// TIA Portal project "S7-1500 ile GELİŞMİŞ Tavuk Çiftliği" (V18)

(* hardware
DEVICE "S7-1500/ET200MP station_1"  S7-1500 station
   slot 0: "Rail_0"  Rack  6ES7 590-1***0-0AA0
   slot 1: "PLC_1"  CPU 1512C-1 PN  6ES7 512-1CK01-0AB0  V2.8
      slot 3: "CPU display_1"  6ES7591-1AA00-0AA0
      slot 32768: "PROFINET interface_1"  X1
         slot 32769: "Port_1"  X1 P1
         slot 32770: "Port_2"  X1 P2
      slot 34817: "Virtual CP interface port_1"  Virtual CP interface port  Virtual CP interface port
DEVICE "HMI_1"  KTP700 Basic PN
   slot 0: "HMI_1"  KTP700 Basic PN  6AV2 123-2GB03-0AX0  14.0.1.0
   slot 1: "HMI_RT_1"  KTP700 Basic PN  6AV2 123-2GB03-0AX0  14.0.1.0
   slot 5: "HMI_1.IE_CP_1"  PROFINET Interface  14.0.1.0
      slot 1: "PROFINET Interface_1"  PROFINET Interface
         slot 1: "Port_1"  Port
*)

// ===== PLC "PLC_1"  CPU 1512C-1 PN =====

VAR_GLOBAL   // PLC tag table "Default tag table"
   "Analog Giriş" AT %IW126 : Word;
   "Kış" AT %I0.1 : Bool;
   "Yaz" AT %I0.2 : Bool;
   "Reset" AT %I0.0 : Bool;
   "Isıtıcı" AT %Q0.1 : Bool;
   "Soğutucu" AT %Q0.2 : Bool;
   "Tag_1" AT %Q0.0 : Bool;
   "yardımcı ısıtıcı" AT %Q0.3 : Bool;
   "yardımcı fan" AT %Q0.4 : Bool;
   "Analog Yardımcı" AT %MW126 : Word;
   "sayaç_1" AT %MD10 : DWord;
   "sayaç_2" AT %MW20 : Int;
   "Tag_2" AT %M0.1 : Bool;
   "Tag_3" AT %M0.2 : Bool;
   "Tag_4" AT %M0.0 : Bool;
END_VAR

// folder: System blocks/Program resources

DATA_BLOCK "IEC_Timer_0_DB"   // DB1
{ S7_Optimized_Access := 'TRUE' }
AUTHOR : Simatic
FAMILY : IEC
NAME : IEC_TMR
VERSION : 1.0
// stored: InstanceOfName IEC_TIMER
"IEC_TIMER"
BEGIN
END_DATA_BLOCK

DATA_BLOCK "IEC_Timer_0_DB_1"   // DB2
{ S7_Optimized_Access := 'TRUE' }
AUTHOR : Simatic
FAMILY : IEC
NAME : IEC_TMR
VERSION : 1.0
// stored: InstanceOfName IEC_TIMER
"IEC_TIMER"
BEGIN
END_DATA_BLOCK

// folder: (top level)

ORGANIZATION_BLOCK "Main"   // OB1, LAD, ProgramCycle
TITLE = "Main Program Sweep (Cycle)"
{ S7_Optimized_Access := 'TRUE' }
VERSION : 0.1
   VAR_INPUT
      Initial_Call : Bool;   // Initial call of this OB
      Remanence : Bool;   // =True, if remanent data are available
   END_VAR
   VAR_TEMP   // added for the SCL form of the ladder/FBD networks
      _w1 : Bool;
   END_VAR
BEGIN

REGION Network 1: Analog girişten alınan değeri okumak içindir.
   // 0-40 derece arası ölçüm yapacak.
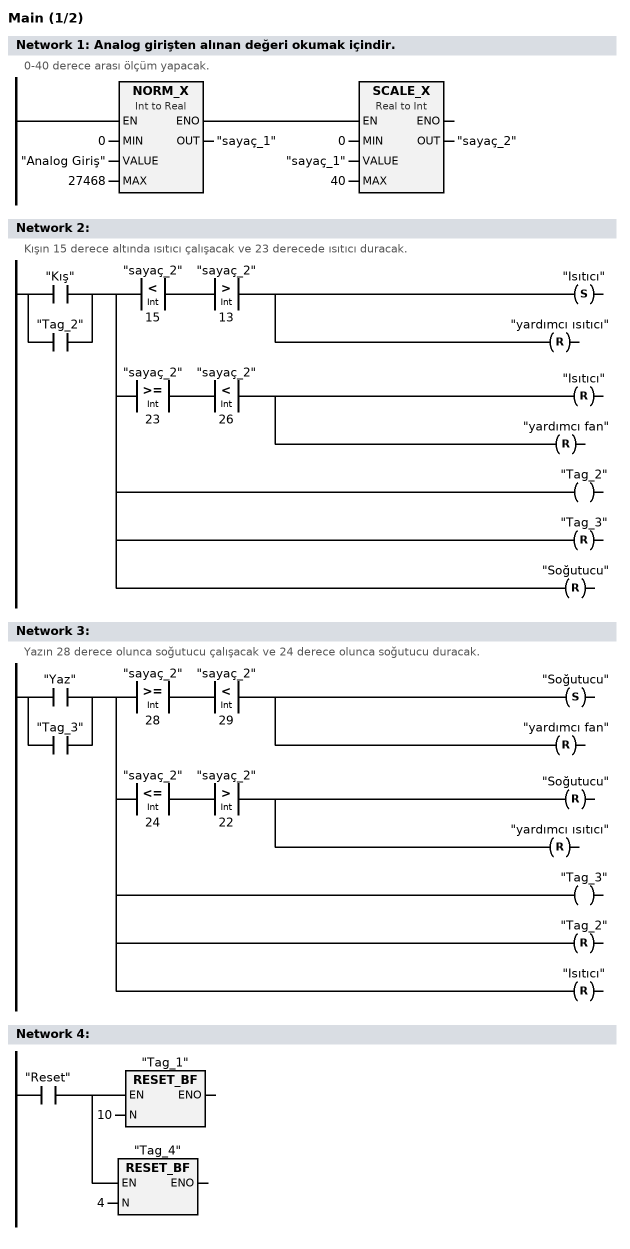
   RUNG wire#powerrail
      { S7_Templates := "[SrcType := Int, DestType := Real]" } Normalize(min := 0, value := "Analog Giriş", max := 27468, out => "sayaç_1")
      { S7_Templates := "[SrcType := Real, DestType := Int]" } Scale(min := 0, value := "sayaç_1", max := 40, out => "sayaç_2")
   END_RUNG
   // the same network as SCL:
   "sayaç_1" := NORM_X(MIN := 0, VALUE := "Analog Giriş", MAX := 27468);
   "sayaç_2" := SCALE_X(MIN := 0, VALUE := "sayaç_1", MAX := 40);
END_REGION

REGION Network 2
   // Kışın 15 derece altında ısıtıcı çalışacak ve 23 derecede ısıtıcı duracak.
   RUNG wire#powerrail
      Contact( "Kış" )
      wire#w1
      { S7_Templates := "SrcType := Int" } LT_Contact(in1 := "sayaç_2", in2 := 15)
      { S7_Templates := "SrcType := Int" } GT_Contact(in1 := "sayaç_2", in2 := 13)
      wire#w2
      S_Coil( "Isıtıcı" )
   END_RUNG
   RUNG wire#powerrail
      Contact( "Tag_2" )
   END_RUNG wire#w1
   RUNG wire#w2
      R_Coil( "yardımcı ısıtıcı" )
   END_RUNG
   RUNG wire#w1
      { S7_Templates := "SrcType := Int" } GE_Contact(in1 := "sayaç_2", in2 := 23)
      { S7_Templates := "SrcType := Int" } LT_Contact(in1 := "sayaç_2", in2 := 26)
      wire#w3
      R_Coil( "Isıtıcı" )
   END_RUNG
   RUNG wire#w3
      R_Coil( "yardımcı fan" )
   END_RUNG
   RUNG wire#w1
      Coil( "Tag_2" )
   END_RUNG
   RUNG wire#w1
      R_Coil( "Tag_3" )
   END_RUNG
   RUNG wire#w1
      R_Coil( "Soğutucu" )
   END_RUNG
   // the same network as SCL:
   #_w1 := "Kış" OR "Tag_2";
   IF #_w1 AND ("sayaç_2" < 15) AND ("sayaç_2" > 13) THEN
       "Isıtıcı" := TRUE;
       "yardımcı ısıtıcı" := FALSE;
   END_IF;
   IF #_w1 AND ("sayaç_2" >= 23) AND ("sayaç_2" < 26) THEN
       "Isıtıcı" := FALSE;
       "yardımcı fan" := FALSE;
   END_IF;
   "Tag_2" := #_w1;
   IF #_w1 THEN
       "Tag_3" := FALSE;
       "Soğutucu" := FALSE;
   END_IF;
END_REGION

REGION Network 3
   // Yazın 28 derece olunca soğutucu çalışacak ve 24 derece olunca soğutucu duracak.
   RUNG wire#powerrail
      Contact( "Yaz" )
      wire#w1
      { S7_Templates := "SrcType := Int" } GE_Contact(in1 := "sayaç_2", in2 := 28)
      { S7_Templates := "SrcType := Int" } LT_Contact(in1 := "sayaç_2", in2 := 29)
      wire#w2
      S_Coil( "Soğutucu" )
   END_RUNG
   RUNG wire#powerrail
      Contact( "Tag_3" )
   END_RUNG wire#w1
   RUNG wire#w2
      R_Coil( "yardımcı fan" )
   END_RUNG
   RUNG wire#w1
      { S7_Templates := "SrcType := Int" } LE_Contact(in1 := "sayaç_2", in2 := 24)
      { S7_Templates := "SrcType := Int" } GT_Contact(in1 := "sayaç_2", in2 := 22)
      wire#w3
      R_Coil( "Soğutucu" )
   END_RUNG
   RUNG wire#w3
      R_Coil( "yardımcı ısıtıcı" )
   END_RUNG
   RUNG wire#w1
      Coil( "Tag_3" )
   END_RUNG
   RUNG wire#w1
      R_Coil( "Tag_2" )
   END_RUNG
   RUNG wire#w1
      R_Coil( "Isıtıcı" )
   END_RUNG
   // the same network as SCL:
   #_w1 := "Yaz" OR "Tag_3";
   IF #_w1 AND ("sayaç_2" >= 28) AND ("sayaç_2" < 29) THEN
       "Soğutucu" := TRUE;
       "yardımcı fan" := FALSE;
   END_IF;
   IF #_w1 AND ("sayaç_2" <= 24) AND ("sayaç_2" > 22) THEN
       "Soğutucu" := FALSE;
       "yardımcı ısıtıcı" := FALSE;
   END_IF;
   "Tag_3" := #_w1;
   IF #_w1 THEN
       "Tag_2" := FALSE;
       "Isıtıcı" := FALSE;
   END_IF;
END_REGION

REGION Network 4
   // no SCL statement known for RBitfield: written as a call
   #_w1 := "Reset";
   IF #_w1 THEN
       RESET_BF(operand := "Tag_1", n := 10);
       RESET_BF(operand := "Tag_4", n := 4);
   END_IF;
END_REGION

REGION Network 5
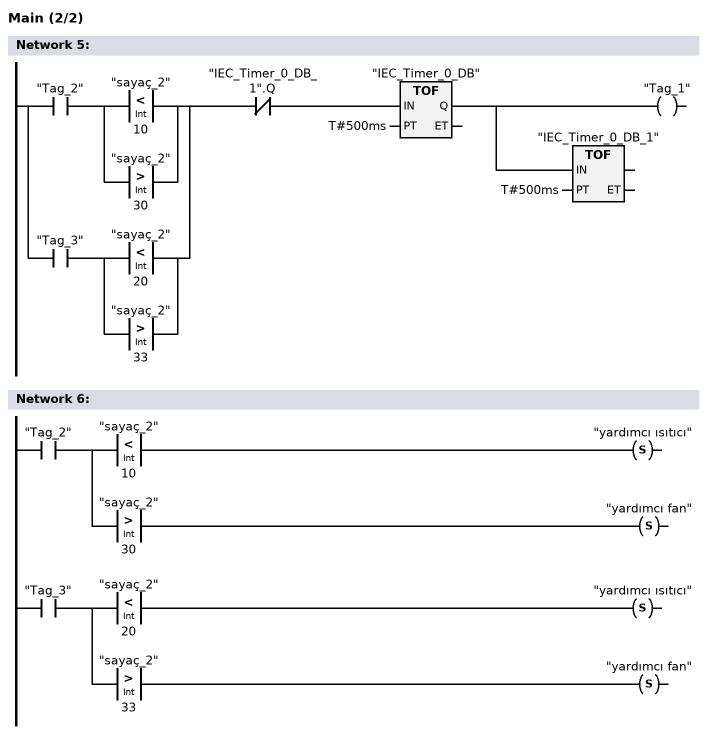
   "IEC_Timer_0_DB".TOF(IN := (("Tag_2" AND (("sayaç_2" < 10) OR ("sayaç_2" > 30))) OR ("Tag_3" AND (("sayaç_2" < 20) OR ("sayaç_2" > 33)))) AND NOT "IEC_Timer_0_DB_1".Q,
                        PT := T#500ms);
   "Tag_1" := "IEC_Timer_0_DB".Q;
   "IEC_Timer_0_DB_1".TOF(IN := "IEC_Timer_0_DB".Q, PT := T#500ms);
END_REGION

REGION Network 6
   RUNG wire#powerrail
      Contact( "Tag_2" )
      wire#w1
      { S7_Templates := "SrcType := Int" } LT_Contact(in1 := "sayaç_2", in2 := 10)
      S_Coil( "yardımcı ısıtıcı" )
   END_RUNG
   RUNG wire#w1
      { S7_Templates := "SrcType := Int" } GT_Contact(in1 := "sayaç_2", in2 := 30)
      S_Coil( "yardımcı fan" )
   END_RUNG
   RUNG wire#powerrail
      Contact( "Tag_3" )
      wire#w2
      { S7_Templates := "SrcType := Int" } LT_Contact(in1 := "sayaç_2", in2 := 20)
      S_Coil( "yardımcı ısıtıcı" )
   END_RUNG
   RUNG wire#w2
      { S7_Templates := "SrcType := Int" } GT_Contact(in1 := "sayaç_2", in2 := 33)
      S_Coil( "yardımcı fan" )
   END_RUNG
   // the same network as SCL:
   IF "Tag_2" AND ("sayaç_2" < 10) THEN "yardımcı ısıtıcı" := TRUE; END_IF;
   IF "Tag_2" AND ("sayaç_2" > 30) THEN "yardımcı fan" := TRUE; END_IF;
   IF "Tag_3" AND ("sayaç_2" < 20) THEN "yardımcı ısıtıcı" := TRUE; END_IF;
   IF "Tag_3" AND ("sayaç_2" > 33) THEN "yardımcı fan" := TRUE; END_IF;
END_REGION
END_ORGANIZATION_BLOCK

(* ===== HMI "HMI_RT_1" =====
system functions are stored by id; their names below are inferred from use
connection "Connection_1": ETHERNET, SMART_S7_1500_OMS
connection "HMI_Connection_1": ETHERNET, SMART_S7_1500_OMS

HMI tags "Default tag table"
   "Tag_ScreenNumber" : UInt, internal
   "sayaç_2" : Int = PLC sayaç_2 AT %MW20, 100 ms
   "Kış" : Bool = PLC Kış AT %I0.1, 100 ms
   "Yaz" : Bool = PLC Yaz AT %I0.2, 100 ms
   "Reset" : Bool = PLC Reset AT %I0.0, 100 ms
   "Tag_3" : Bool = PLC Tag_3 AT %M0.2, 100 ms
   "Tag_2" : Bool = PLC Tag_2 AT %M0.1, 100 ms
   "Soğutucu" : Bool = PLC Soğutucu AT %Q0.2, 100 ms
   "Isıtıcı" : Bool = PLC Isıtıcı AT %Q0.1, 100 ms
   "uyarı" : Bool = PLC Tag_1 AT %Q0.0, 100 ms
   "yardımcı ısıtıcı" : Bool = PLC "yardımcı ısıtıcı" AT %Q0.3, 100 ms
   "yardımcı fan" : Bool = PLC "yardımcı fan" AT %Q0.4, 100 ms

graphic list "yaz": 0 ''; 1 'Graphic_26'

graphic list "kış1": 0 ''; 1 'Graphic_28'

graphic list "kış2": 0 ''; 1 'Graphic_27'

graphic list "fan": 0 'Graphic_30'; 1 'Graphic_31'

graphic list "ısıtıcı": 0 'Graphic_32'; 1 'Graphic_33'

graphic list "uyarı": 0 'Graphic_36'; 1 'Graphic_15'

graphic list "yardımcı ısıtıcı": 0 'Graphic_32'; 1 'Graphic_33'

graphic list "yardımcı fan": 0 'Graphic_38'; 1 'Graphic_37'

Template "Template_1" 800x480
   Button "Exit" at 714,429 size 71x50; TextOff 'Exit'; PictureOff "ExitRuntime_KTP700_Basic_PN_TR"; PictureOn "ExitRuntime_KTP700_Basic_PN_TR"
      on Release: StopRuntime(0)
   Button "Language" at 614,429 size 71x50; TextOff 'Language'; PictureOff "ToggleLanguage_KTP700_Basic_PN_TR"; PictureOn "ToggleLanguage_KTP700_Basic_PN_TR"
      on Release: function_fb9197e8(-1)
   Button "Log on" at 514,429 size 71x50; TextOff 'Log on'; PictureOff "Login_KTP700_Basic_PN_TR"; PictureOn "Login_KTP700_Basic_PN_TR"
      on Release: function_a2a04561()
   Button "Alarms" at 114,429 size 71x50; TextOff 'Alarms'; PictureOff "AlarmDisplay_KTP700_Basic_PN_TR"; PictureOn "AlarmDisplay_KTP700_Basic_PN_TR"
      on Release: function_ef3f5d25("Alarm window_Unacknowledged", -1)
   Button "Start screen" at 14,429 size 71x50; TextOff 'Start screen'; PictureOff "NavigateHome_KTP700_Basic_PN_TR"; PictureOn "NavigateHome_KTP700_Basic_PN_TR"
      on Release: ActivateScreen("Root screen", 0)
   SymbolicIOField "Symbolic_IO_Field_Screen" at 93,9 size 600x33; TextOff '0'; TextOn '1'; TextList "TextList_ScreenNames"
      ProcessValue <- "Tag_ScreenNumber"
      on Change: ActivateScreenByNumber("Tag_ScreenNumber", 0)
   DateTimeField "HmiScreenItemData" at 695,25 size 105x25
   DateTimeField "HmiScreenItemData_1" at 695,0 size 105x25
   GraphicView "Logo" at 0,0 size 91x51; Picture "Logo of HMI_1"

screen "Root screen" 800x480, template "Template_1"
   on GenerateScreen: SetTag("Tag_ScreenNumber", 1)
   Button "Button_2" at 170,273 size 96x57; TextOff 'Kış'
      on Press: SetBit("Kış")
      on Release: ResetBit("Kış")
   Button "Button_3" at 170,337 size 96x57; TextOff 'Yaz'
      on Release: ResetBit("Yaz")
      on Press: SetBit("Yaz")
   Button "Button_4" at 170,210 size 96x56; TextOff 'Reset'
      on Press: SetBit("Reset")
      on Release: ResetBit("Reset")
   IOField "I/O field_1" at 170,144 size 96x60; FormatPattern s99999
      ProcessValue <- "sayaç_2"
   Bar "Bar_1" at 279,144 size 104x252; MinimumValue 0; MaximumValue 40
      ProcessValue <- "sayaç_2"
   GraphicIOField "Graphic I/O field_1" at 42,277 size 96x48; PictureList "kış1"
      ProcessValue <- "Tag_2"
   GraphicIOField "Graphic I/O field_2" at 42,325 size 96x48; PictureList "kış2"
      ProcessValue <- "Tag_2"
   GraphicIOField "Graphic I/O field_3" at 42,172 size 96x80; PictureList "yaz"
      ProcessValue <- "Tag_3"
   GraphicIOField "Graphic I/O field_4" at 416,278 size 133x100; PictureList "ısıtıcı"
      ProcessValue <- "Isıtıcı"
   GraphicIOField "Graphic I/O field_5" at 414,144 size 135x109; PictureList "fan"
      ProcessValue <- "Soğutucu"
   GraphicView "Graphic view_2" at 182,62 size 74x76; Picture "Graphic_34"
      Visibility <- "uyarı"
   GraphicView "Graphic view_3" at 677,53 size 123x60; Picture "Graphic_35"
   GraphicIOField "Graphic I/O field_6" at 279,66 size 104x78; PictureList "uyarı"
      ProcessValue <- "uyarı"
   GraphicIOField "Graphic I/O field_7" at 567,145 size 132x107; PictureList "yardımcı fan"
      ProcessValue <- "yardımcı fan"
   GraphicIOField "Graphic I/O field_8" at 567,279 size 132x100; PictureList "yardımcı ısıtıcı"
      ProcessValue <- "yardımcı ısıtıcı"
   TextField "Text field_1" at 444,124 size 87x23; Text 'Ana Isıtıcı'
   TextField "Text field_2" at 567,256 size 126x23; Text 'Yardımcı Isıtıcı'
   TextField "Text field_3" at 424,254 size 117x23; Text 'Ana Soğutucu'
   TextField "Text field_4" at 555,124 size 156x23; Text 'Yardımcı Soğutucu'
*)